// TIA Portal V17 export
// export: Created 2024-09-02T12:50:24.3943373Z, ExportSetting WithDefaults, DisplayName Totally Integrated Automation Portal, DisplayVersion V17, DisplayName TIA Portal Openness, DisplayVersion V17, DisplayName TIA Portal Version Control Interface, DisplayVersion V17, DisplayName STEP 7 Professional, DisplayVersion V17, DisplayName STEP 7 Safety, DisplayVersion V17, DisplayName WinCC Professional, DisplayVersion V17
DATA_BLOCK "DBi_MES_StationStatus_OP70"   // DB704
{ S7_Optimized_Access := 'FALSE' }
VERSION : 0.1
// stored: AutoNumber false, DBAccessibleFromOPCUA true, IsOnlyStoredInLoadMemory false, IsWriteProtectedInAS false
   VAR
      StatusStation : Struct
         WsState { ExternalWritable := 'False'} : Int;
         AutomaticMode { ExternalWritable := 'False'} : Bool;
         Starved { ExternalWritable := 'False'} : Bool;
         Blocked { ExternalWritable := 'False'} : Bool;
         ManualMode { ExternalWritable := 'False'} : Bool;
         Fault { ExternalWritable := 'False'} : Bool;
         FrequencialControlProgress : Bool;
         ChangeToolInProgress : Bool;
         PartMissing : Bool;
         AndonCall : Bool;
         Maintenance : Bool;
         Quality : Bool;
         Proces : Bool;
         ErrorCode { ExternalWritable := 'False'} : Int;
      END_STRUCT;
      ErrorCode : Int;
      Users : Struct
         level : Int;
      END_STRUCT;
      init : Struct
         StatusStation : Struct
            WsState : Int;
            AutomaticMode : Bool;
            Starved : Bool;
            Blocked : Bool;
            ManualMode : Bool;
            Fault : Bool;
            FrequencialControlProgress : Bool;
            ChangeToolInProgress : Bool;
            PartMissing : Bool;
            AndonCall : Bool;
            Maintenance : Bool;
            Quality : Bool;
            Proces : Bool;
            ErrorCode : Int;
         END_STRUCT;
         ErrorCode : Int;
         Users : Struct
            level : Bool;
         END_STRUCT;
      END_STRUCT;
   END_VAR
BEGIN
END_DATA_BLOCK
